{attribute addProperty BoxType "AT2020-0250-0019"}
{attribute addProperty Id "A_0085_AT2050_5500_0018_AT2050_5500AT2050_3DCFC8D064080"}
{attribute addProperty CRC "3520646050"}
{attribute addProperty SizeInBites "640"}
{attribute addProperty SizeInBytes "80"}
TYPE A_0060_AT2020_0250_0019_AT2020_0250_D1D8CBA2 EXTENDS AT2020_9506A482 :
STRUCT
	{attribute addProperty Name "A_0085_AT2050_5500_0018_AT2050_5500"}
	A_0085_AT2050_5500_0018_AT2050_5500 : AT2050_3DCFC8D0;
END_STRUCT
END_TYPE

(* stored: Version 1.2.0.0, ProductVersion 3.1.4024.9
   DUT A_0060_AT2020_0250_0019_AT2020_0250_D1D8CBA2: Id {9bcba79b-d6a6-4c1a-a360-9b32616f5f5c} *)
